PROGRAM MAIN
VAR CONSTANT
	IGNORE_DEFINITION: BOOL := TRUE;
END_VAR
VAR
	m_errorManager: ErrorManager;
	m_services: ServiceContainer(ADR(m_errorManager));
	
	m_panelMgr: PanelManager(
		m_services.PtrStateTracker,
		EProcessVariables.Pnl_Stack_Start,
		0,
		EProcessVariables.Pnl_Stack_Mode,
		EProcessVariables.Pnl_Stack_EStop,
		0);
	
	// instantiate machine behavior model
	m_container: HardwareContainer(
		m_services.PtrStateTracker, 
		m_services.PtrProcessManager, 
		ADR(m_errorManager));
	
	m_modes: MachineModes(ADR(m_services), ADR(m_panelMgr));
	
	m_appObservation: ARRAY[EProcessVariables.OpMode_Stack..EProcessVariables.OpMode_Stack] OF SValue;

	// TESTING
// 	m_lscConnected: BOOL;
// 	m_craneConnected: BOOL;
// 	m_stackConnected: BOOL;
// 	m_stampConnected: BOOL;
END_VAR

// process state observation
m_appObservation[EProcessVariables.OpMode_Stack].DataType := EDataType.string_t;
m_appObservation[EProcessVariables.OpMode_Stack].Value.String_t := m_modes.SFCCurrentStep;
m_appObservation[EProcessVariables.OpMode_Stack].Defined := TRUE;

// cylic service updates
m_services.PtrStateTracker^.CyclicUpdateStatus(IGNORE_DEFINITION, m_appObservation);
m_services.PtrProcessManager^.CyclicManageBehavior();

// main state machine
m_modes();

// TESTING
// IF m_services.PtrStateTracker^.GetString(EProcessVariables.OpMode_LSC) <> '' THEN
// 	m_lscConnected := TRUE;
// END_IF
// IF m_services.PtrStateTracker^.GetString(EProcessVariables.OpMode_Stack) <> '' THEN
// 	m_stackConnected := TRUE;
// END_IF
// IF m_services.PtrStateTracker^.GetString(EProcessVariables.OpMode_Stamp) <> '' THEN
// 	m_stampConnected := TRUE;
// END_IF
// IF m_services.PtrStateTracker^.GetString(EProcessVariables.OpMode_Crane) <> '' THEN
// 	m_craneConnected := TRUE;
// END_IF

END_PROGRAM

(* stored: Version 1.1.0.1
   POU MAIN: Id {189c3a67-5245-4ff4-9cf5-6680f225c565}, SpecialFunc None *)
